// TwinCAT 3 PLC project PLC
// ProgramVersion: 3.1.4026.19
// libraries:
//   SPT Base Types, * (Beckhoff Automation LLC)
//   SPT Components, * (Beckhoff Automation LLC)
//   SPT Diagnostic, * (Beckhoff Automation LLC)
//   SPT EtherCat, * (Beckhoff Automation LLC)
//   SPT Event Logger, * (Beckhoff Automation LLC)
//   SPT Motion Control, * (Beckhoff Automation LLC)
//   SPT Utilities, * (Beckhoff Automation LLC)
//   Tc2_MC2, * (Beckhoff Automation GmbH)
//   Tc2_Standard, * (Beckhoff Automation GmbH)
//   Tc2_System, * (Beckhoff Automation GmbH)
//   Tc3_EventLogger, * (Beckhoff Automation GmbH)
//   Tc3_Module, * (Beckhoff Automation GmbH)
//   Tc3_PackML_V3, * (Beckhoff Automation GmbH)
// project tree:
//   / GlobalTextList.TcGTLO, PlcTask.TcTTO, Visualization Manager.TcVMO (not stored)
//   POUs/Function Blocks/ FB_HomeRoutine_CalibrationCam.TcPOU
//   POUs/ MAIN.TcPOU
//   POUs/Modules/00 Machine/ Machine.TcPOU
//   VISUs/ Visualization.TcVIS
// real-time tasks:
//   TASK PlcTask: cycle T#10ms, priority 20, ADS port 350
// motion (NC):
// variable links:
//   PLC/PLC Instance <-> NC-Task 1 SAF/Axes/Axis 1
//     PlcTask Inputs/MAIN.Machine.VAxis.BasicAxis._Axis.NcToPlc <-> Outputs/ToPlc
//     PlcTask Outputs/MAIN.Machine.VAxis.BasicAxis._Axis.PlcToNc <-> Inputs/FromPlc

CONFIGURATION PLC
    RESOURCE PLC ON TwinCAT3
        TASK PlcTask(INTERVAL := T#10ms, PRIORITY := 20);
        PROGRAM MAIN WITH PlcTask : MAIN;
    END_RESOURCE
END_CONFIGURATION

// ---- POUs/MAIN.TcPOU
PROGRAM MAIN
VAR
	Machine : Machine := (Name := 'Machine');
END_VAR

(*All sample code provided by Beckhoff Automation LLC are for illustrative purposes only and are provided “as is” and without any warranties, express or implied. Actual implementations in applications will vary significantly. Beckhoff Automation LLC shall have no liability for, and does not waive any rights in relation to, any code samples that it provides or the use of such code samples for any purpose.*)

(*
	The FB_Component_BasicAxis within the SPT Components library is configured to use a Homing Routine defined in the SPT_MotionControl library.
	FB_HomeRoutine_SetZeroHere, which is an implementation of the MC_SetPosition from the Tc2_MC2 library. 
	The strategy design pattern is used for HomeMethod, ResetMethod, and ExternalSequence. 
	You can change the default homing routine by declaring an instance of a function block that implements the interface I_MotionSequence, 
	and then passing it to the HomeMethod property of your instance of FB_Component_BasicAxis. 
	Within the SPT Motion Control library we provide three other homing options (FB_HomeRoutine_AbsHoming, FB_HomeRoutine_HardStop, FB_HomeRoutine_SetPosition). 
	Further documentation can be found here: https://beckhoff-usa-community.github.io/SPT-Libraries/SPT_MotionControl/functionblocks.html#home-routines
	
	For this sample project an Axis Component is declared within FB_Machine.
	In the Execute method of FB_Machine one of 4 possible home routines can be selected.
	The first 3 are from the SPT Motion Control library, and the fourth is availble in the project.
	
	Use the Visu to move tha state machine into Execute
	and then toggle one of the four home routines in the execute mehod to start the homing process.
	When using HomeCalCam, you will need to toggle _CalibrationCam within the FB_HomeRoutine_CalibrationCam
	to simulate the axis moving onto and off of a physical home switch.
 	A Maintained PB has been added to the Visu for the _CalibrationCam
*)

//This is for debug only and should be removed
_AppInfo.KeepOutputsOnBP := TRUE;

//
Machine.CyclicLogic();

END_PROGRAM

// ---- POUs/Modules/00 Machine/Machine.TcPOU
FUNCTION_BLOCK Machine EXTENDS FB_PackML_BaseModule
VAR
	VAxis	  : FB_Component_BasicAxis := (Name := 'V Axis');
	AxisHomed : BOOL;

	//Home Commands
	HomeAbs		 : BOOL;
	HomeHardStop : BOOL;
	HomeSetPos	 : BOOL;
	HomeCalCam	 : BOOL;

	//Homing Options
	AbsHoming	   : FB_HomeRoutine_AbsHoming;
	HardStopHoming : FB_HomeRoutine_HardStop;
	SetPosition	   : FB_HomeRoutine_SetPosition;
	CalibrationCam : FB_HomeRoutine_CalibrationCam;
END_VAR

// This method serves as the entry point for all underlying FB logic
METHOD PUBLIC CyclicLogic

// This method should be called cyclically by descendant function blocks by invoking SUPER^.CyclicLogic().  Alternatively, the contents of this method could be reimplemented entirely in which case a call to this method would not be necessary.
IF NOT _InitComplete THEN
	_InitComplete := Initialize();
	RETURN;
END_IF

SUPER^.CyclicLogic();
END_METHOD

// This method contains code which will execute when this PackML module is in the Execute state
METHOD PROTECTED Execute

// The base implementation of this method is empty. User must override this method to provide functionality.

// This method is called as required by StateControl()
CASE SequenceState OF
	0:
		IF HomeAbs THEN
			HomeAbs			 := FALSE;
			VAxis.HomeMethod := AbsHoming;
			SequenceState	 := SequenceState + 10;
		END_IF

		IF HomeHardStop THEN
			HomeHardStop	 := FALSE;
			VAxis.HomeMethod := HardStopHoming;
			SequenceState	 := SequenceState + 10;
		END_IF

		IF HomeSetPos THEN
			HomeSetPos		 := FALSE;
			VAxis.HomeMethod := SetPosition;
			SequenceState	 := SequenceState + 10;
		END_IF

		IF HomeCalCam THEN
			HomeCalCam		 := FALSE;
			VAxis.HomeMethod := CalibrationCam;
			SequenceState	 := SequenceState + 10;
		END_IF

	10:
		IF VAxis.Home() THEN
			SequenceState := SequenceState + 10;
		END_IF

	20:
		IF VAxis.Axis.Status.Homed THEN
			SequenceState := SequenceState + 10;
		END_IF

	30:
		AxisHomed := TRUE;
END_CASE
END_METHOD

// Automatically enables and disables HMI control based on the PackML mode
METHOD PROTECTED HMIPermissions

// This method is called cyclically by CyclicLogic()
AllowHMIControl(ThisModuleOnly := TRUE);
END_METHOD

//  Basic module initialization logic
METHOD PROTECTED Initialize : BOOL;

// This method is called by CyclicLogic() as required
Initialize := FALSE;
CASE DescendantSequenceState OF
	0:
		RegisterComponent(Component := VAxis);
		DescendantSequenceState := DescendantSequenceState + 10;

	10:
		IF SUPER^.Initialize() THEN
			Initialize := TRUE;
		END_IF
END_CASE
END_METHOD

// This method contains code which will execute when this PackML module is in the Starting state
METHOD PROTECTED Starting

// This method is called as required by StateControl()
CASE SequenceState OF
	0:
		NoStateTasksToComplete := FALSE;
		SequenceState		   := SequenceState + 10;

	10:
		IF VAxis.Enable() THEN
			SequenceState := SequenceState + 10;
		END_IF

	20:
		IF VAxis.Enabled THEN
			SequenceState := SequenceState + 10;
		END_IF

	30:
		StateTasksComplete := TRUE;
END_CASE

SUPER^.Starting();
END_METHOD

END_FUNCTION_BLOCK

// ---- POUs/Function Blocks/FB_HomeRoutine_CalibrationCam.TcPOU
FUNCTION_BLOCK FB_HomeRoutine_CalibrationCam EXTENDS FB_CyclicFB IMPLEMENTS I_MotionSequence
VAR
	_Axis : I_BasicAxis;

	//
	MCHomeCalCam	: MC_Home;
	_HomingDn		: BOOL;
	SequenceStep	: UDINT;
	_Position		: LREAL;
	_Options		: ST_HomingOptions;
	_CalibrationCam : BOOL;
END_VAR

PROPERTY Axis : I_BasicAxis
GET
Axis := _Axis;
END_GET
SET
_Axis := Axis;
END_SET
END_PROPERTY

PROPERTY CalibrationCam : BOOL
GET
CalibrationCam := _CalibrationCam;
END_GET
SET
_CalibrationCam := CalibrationCam;
END_SET
END_PROPERTY

METHOD PUBLIC CyclicLogic
CASE SequenceStep OF
	10:
		IF _Axis <> 0 THEN
			MCHomeCalCam(Axis			 := _Axis.Axis,
						 Execute		 := TRUE,
						 Position		 := _Position,
						 HomingMode		 := MC_HomingMode.MC_DefaultHoming,
						 Options		 := _Options,
						 bCalibrationCam := _CalibrationCam);

			IF NOT MCHomeCalCam.Busy THEN
				IF MCHomeCalCam.Error THEN
					_Error		 := TRUE;
					_ErrorID	 := MCHomeCalCam.ErrorID;
					SequenceStep := 0;
				ELSE
					//No error occurred
					SequenceStep := 0;
				END_IF

				MCHomeCalCam(Axis := _Axis.Axis, Execute := FALSE);
			END_IF
		END_IF
END_CASE

_Busy := SequenceStep <> 0;
END_METHOD

METHOD Execute : BOOL
IF (_Axis = 0) OR _Busy THEN
	RETURN;
END_IF

_Busy		 := TRUE;
_Error		 := FALSE;
_ErrorID	 := 0;
_HomingDn	 := FALSE;
SequenceStep := 10;
Execute		 := TRUE;
END_METHOD

PROPERTY Options : ST_HomingOptions
GET
Options := _Options;
END_GET
SET
_Options := Options;
END_SET
END_PROPERTY

PROPERTY Position : LREAL
GET
Position := _Position;
END_GET
SET
_Position := Position;
END_SET
END_PROPERTY

END_FUNCTION_BLOCK

// ---- GlobalTextList.TcGTLO
TEXTLIST GlobalTextList
  232 = 'Calibration Cam Switch'
END_TEXTLIST

// ---- VISUs/Visualization.TcVIS
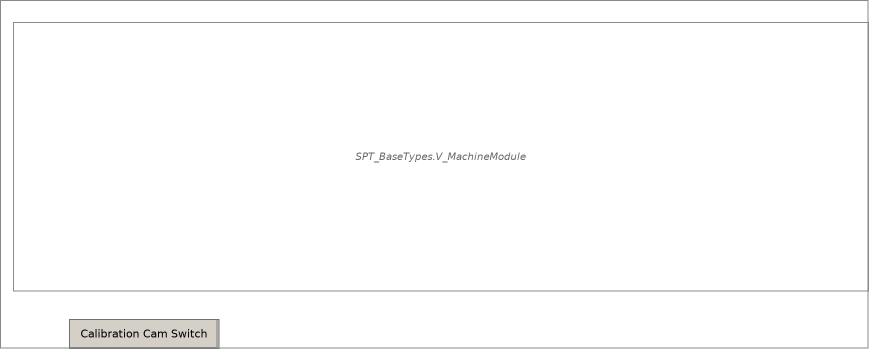
VISUALIZATION Visualization  // 869x349
    Frame (13,22 856x269)
        shows SPT_BaseTypes.V_MachineModule(HMI := MAIN.Machine.PackMLBaseModule_HMI)
    Button (69,319 150x30), "Calibration Cam Switch"
        toggle MAIN.Machine.CalibrationCam._CalibrationCam
END_VISUALIZATION
